FUNCTION_BLOCK FB_ExternalControl
VAR

END_VAR
VAR
END_VAR

END_FUNCTION_BLOCK

(* stored: Version 1.1.0.1, ProductVersion 3.1.4024.12
   POU FB_ExternalControl: Id {8e859215-c51a-4c77-a474-4ba070448a0e}, SpecialFunc None *)
